FUNCTION_BLOCK FB_State_Idle EXTENDS FB_BaseState IMPLEMENTS Istate
VAR_INPUT
END_VAR
VAR_OUTPUT
END_VAR
VAR
END_VAR

METHOD mStart
ADSLOGSTR(ADSLOG_MSGTYPE_HINT, 'Start signal asserted.', '');
END_METHOD

{error 'add property implementation or delete property to use base implementation'}
PROPERTY pMessage : STRING
GET
pMessage := 'Waiting for start signal';
END_GET
END_PROPERTY

END_FUNCTION_BLOCK

(* stored: Version 1.1.0.1, ProductVersion 3.1.4024.9
   POU FB_State_Idle: Id {611356df-394d-4c5b-b921-ec2aaa8026ea}, SpecialFunc None
   Method mStart: Id {e0f33d6c-00a6-4167-a8f6-932d36b0108d}
   Property pMessage: Id {d890618a-09b3-43e9-afab-a6a1fc2446d2}
   Get Get: Id {d2de0552-adcd-4843-bfaa-36361f39a9cf} *)
